TYPE T_Ctrl_SIf_DRV_Cur :
STRUCT
	dinPulseCounter: DINT;
	dinPos_um: DINT;
	dinSpeed_um_s: DINT;
END_STRUCT
END_TYPE

(* stored: Version 1.1.0.1, ProductVersion 3.1.0.19
   DUT T_Ctrl_SIf_DRV_Cur: Id {59e3857f-8003-4339-801b-51d7e76ff3a7} *)
